//{{V2}}
ORGANIZATION_BLOCK OB1
TITLE= "Zyklisches Hauptprogramm"


AUTHOR:nb
FAMILY:nb
NAME:nb
VERSION:1.0


VAR_TEMP
       OB1_EV_CLASS:BYTE //Bits 0-3 = 1 (Coming event), Bits 4-7 = 1 (Event class 1)
       OB1_SCAN_1:BYTE //1 (Cold restart scan 1 of OB 1), 3 (Scan 2-n of OB 1)
       OB1_PRIORITY:BYTE //1 (Priority of 1 is lowest)
       OB1_OB_NUMBR:BYTE //1 (Organization block 1, OB1)
       OB1_RESERVED_1:BYTE //Reserved for system
       OB1_RESERVED_2:BYTE //Reserved for system
       OB1_PREV_CYCLE:INT //Cycle time of previous OB1 scan (milliseconds)
       OB1_MIN_CYCLE:INT //Minimum cycle time of OB1 (milliseconds)
       OB1_MAX_CYCLE:INT //Maximum cycle time of OB1 (milliseconds)
       OB1_DATE_TIME:DATE_AND_TIME //Date and time OB1 started
END_VAR
BEGIN

NETWORK
TITLE=
//{{a}}

       U    E0.0
       FP   M      1000.0
       U(
       L    MW10
       L    10
       <I
       )

       SPBN push

       L    MW12
       L    1
       +I
       T    MW12



       L    MW10
       L    P#        2.0
       *I
       T    MD100


       AUF  DB       10

       L    MW12
       T    DBW [MD100]



       L    MW10
       L    1
       +I
       T    MW10


//       L    "index"
//       L    10
//       MOD
//       T    "index"


push:  NOP  0
NETWORK
TITLE=
//{{a}}

       U    E0.1
       FP   M      1000.1
       U(
       L    MW10
       L    0
       >I
       )
       SPBN pop


       AUF  DB       10


       L    MW10
       L    1
       -I
       T    MW10




//       L    "index"
//       L    10
//       +I
//       L    10
//       MOD
//       T    "index"

       L    MW10
       L    P#        2.0
       *I
       T    MD100



       L    DBW [MD100]
       ITB
       T    AW       10

       L    0
       T    DBW [MD100]



pop:   NOP  0
NETWORK
TITLE=
//{{a}}




END_ORGANIZATION_BLOCK
